(* IEC 61131-3 sources: lc3-wifi-kurs/src/example_8_PID_Test, 1 file *)

(* ---- Program_PID_Test.iecst ---- *)
PROGRAM Program_PID_Test
	VAR
		pid : PID;
	END_VAR

	pid();
END_PROGRAM
